Fanuc KAREL source: kt00484.KL

-- PROVISIONAL review KL for V940-1; original PC SHA256 496e820cf56d33284622033e6a9ed9a37a1354281d9318ef95159041ede35008
-- Incomplete behavior may be omitted. Consult companion uncertainty JSON. Do not deploy.
PROGRAM KT00484
%NOLOCKGROUP
-- UNRESOLVED_DECL P1 type=000101
-- UNRESOLVED_DECL P2 type=000106
-- UNRESOLVED_DECL OUT type=000101
BEGIN
  -- V9_ZERO_TABLE_METADATA_HINT layout=0001; no indexed target words; source/name/runtime held
  -- UNRESOLVED_PC offsets 5-20; opcodes 2E,22,32,35
  -- UNRESOLVED_PC offsets 25-54; opcodes 49,49,7E,60,4A
  -- UNRESOLVED_PC offsets 59-63; opcodes 7F
END KT00484
